# EPICS substitutions: db/Beckhoff_2XXX/ecmcEL2521.substitutions
file "ecmcEcSlave.template"
{
  pattern {}
          {}
}

file "ecmcEL2521.template"
{
  pattern {LINR,    ESLO, EOFF,    EGU,        PREC, LOW, LOLO, HIGH, HIHI, HYST, LLSV,       LSV,        HSV,        HHSV        }
          {"SLOPE", 1,    0,       "Counts",   0,    0,   0,    0,    0,    0,    "NO_ALARM", "NO_ALARM", "NO_ALARM", "NO_ALARM"  }
}
